// TIA Portal V20 export
TYPE "LAxisCtrl_typePosSuperimposed"
TITLE = LAxisCtrl_typePosSuperimposed
// Support: tech.team.motioncontrol@siemens.com 
// Fax: +49 (0) 9131/98-1297
   STRUCT
      distance : LReal := 0.0;   // Distance for superimposed positioning
      velocityDiff : LReal := -1.0;   // Maximum velocity deviation compared to the active motion (Value > 0.0: The specified value is used; Value = 0.0: Not permitted; Value < 0.0: Use of the default value configured in the technology object)
      acceleration : LReal := -1.0;   // Acceleration for positioning (Value > 0.0: The specified value is used; Value = 0.0: Not permitted; Value < 0.0: Use of the default value configured in the technology object)
      deceleration : LReal := -1.0;   // Deceleration for positioning (Value > 0.0: The specified value is used; Value = 0.0: Not permitted; Value < 0.0: Use of the default value configured in the technology object)
      jerk : LReal := -1.0;   // Jerk for positioning (Value > 0.0: Smooth velocity profile, the specified value is used; Value = 0.0: Trapezoid velocity profile; Value < 0.0: Use of the default value configured in the technology object)
      direction : DInt := 0;   // Motion direction of the axis (0: The sign of the distance parameter defines the direction; 1: Positive negative; 2: Negative direction)
   END_STRUCT;
END_TYPE
